# EPICS autosave request: measCompApp/Db/measCompAnalogIn_settings.req
$(P)$(R)Range
$(P)$(R)Mode
$(P)$(R).LOPR
$(P)$(R).HOPR
$(P)$(R).EGUF
$(P)$(R).EGUL
$(P)$(R).PREC
$(P)$(R).SCAN
